FUNCTION SuccessTestFunction : T_MAXSTRING
VAR_INPUT
	foo : T_MAXSTRING;
	hello : T_MAXSTRING;
END_VAR
VAR
END_VAR

SuccessTestFunction := concat(foo, hello);

END_FUNCTION

(* stored: Version 1.1.0.1, ProductVersion 3.1.4024.12
   POU SuccessTestFunction: Id {a12dc10c-a75e-47c2-a1f7-c8979a1e8b02}, SpecialFunc None *)
